{attribute 'qualified_only'}
{attribute 'strict'}
TYPE E_BufferStates :
(
	Init := 0,
	Waiting,
	CheckBuffer,
	FindEmptyLocation,
	InsertIntoBuffer,
	CheckTicekts,
	SetTrafficLightRed,	
	SendOutOfBuffer,
	SetTrafficLightGreen
);
END_TYPE

(* stored: Version 1.1.0.1, ProductVersion 3.1.4024.2
   DUT E_BufferStates: Id {7ee054bf-9136-4bf5-bd28-f5d4d017a2b6} *)
